FUNCTION_BLOCK TestHarness
VAR
	Pass    : UDINT;
    Fail    : UDINT;
    Lines   : ARRAY[1..200] OF STRING(255);
    LineIdx : UDINT;
END_VAR

METHOD AssertTrue : BOOL
VAR_INPUT
	Condition	: BOOL;
	Name		: STRING;
END_VAR
IF Condition THEN
    Logger(CONCAT('PASS: ', Name));
    Pass := Pass + 1;
ELSE
    Logger(CONCAT('FAIL: ', Name));
    Fail := Fail + 1;
END_IF
AssertTrue := Condition;
END_METHOD

METHOD Clear : BOOL
VAR_INPUT
END_VAR
Pass := 0; 
Fail := 0; 
LineIdx := 0;
Clear := TRUE;
END_METHOD

METHOD PRIVATE Logger : BOOL
VAR_INPUT
	StringIn	: STRING;
END_VAR
IF LineIdx < UPPER_BOUND(Lines, 1) THEN
    LineIdx := LineIdx + 1;
    Lines[LineIdx] := StringIn;
END_IF
Logger := TRUE;
END_METHOD

END_FUNCTION_BLOCK

(* stored: Version 1.1.0.1
   POU TestHarness: Id {fe2f4f26-4df0-4adf-910a-6d052233beb9}, SpecialFunc None
   Method AssertTrue: Id {f0f7f023-e373-441a-be94-b2c83ce23265}
   Method Clear: Id {dbe7a9da-87f3-4b93-8561-a31d9c598000}
   Method Logger: Id {d471a513-3a33-4cd9-9d50-b6c9db120c2e} *)
